// Implicitly generated code : DO NOT EDIT
FUNCTION CheckDivLReal : LREAL
VAR_INPUT
	divisor:LREAL;
END_VAR

// Implicitly generated code : Only an Implementation suggestion
{noflow}
Fault_Count_G(CU:=FALSE) ; 
IF divisor = 0 THEN
	CheckDivLReal:=1;
		Fault_Count_G(CU:=TRUE) ; 
ELSE
	CheckDivLReal:=divisor;
END_IF;
{flow}

END_FUNCTION

(* stored: Version 1.1.0.1, ProductVersion 3.1.4024.2
   POU CheckDivLReal: Id {62da009c-5d75-4bd6-889c-d94e781aa52e}, SpecialFunc CheckDivReal64 *)
